// TIA Portal V19 export
ORGANIZATION_BLOCK "CYCL_FLT"   // OB80, STL, TimeErrorInterrupt
TITLE = "Cycle Time Fault"
{ S7_Optimized_Access := 'TRUE' }
VERSION : 0.0
   VAR_INPUT
      Fault_ID : Byte;   // Fault identifier
      Csg_OBnr : OB_ANY;   // Number of OB causing the error
      Csg_Prio : UInt;   // Priority of OB causing the error
   END_VAR
BEGIN
END_ORGANIZATION_BLOCK
